// TIA Portal V17 export
// export: Created 2025-03-10T13:11:55.1694581Z, ExportSetting WithDefaults, DisplayName Totally Integrated Automation Portal, DisplayVersion V17 Update 8, DisplayName TIA Portal Openness, DisplayVersion V17 Update 8, DisplayName TIA Portal Version Control Interface, DisplayVersion V17, DisplayName SINAMICS Startdrive Advanced, DisplayVersion V17 SP2, DisplayName SINAMICS Startdrive G110M, G120, G120C, G120D, G120P, G115D, DisplayVersion V17 SP2, DisplayName SINAMICS Startdrive G130, G150, S120, S150, SINAMICS MV, S210, DisplayVersion V17 SP2, DisplayName STEP 7 Professional, DisplayVersion V17 Update 8, DisplayName SINUMERIK ONE STEP 7 Toolbox, DisplayVersion V17 Update 12, DisplayName SINUMERIK 840D sl STEP 7 Toolbox, DisplayVersion V17 Update 12, DisplayName STEP 7 Safety, DisplayVersion V17 Update 6, DisplayName WinCC Advanced, DisplayVersion V17 Update 8
TYPE "LBP_typeTMLoadMT"
TITLE = Tool management / Gestión de herramientas / Werkzeugverwaltung
// User data type for block LBP_TMLoadMT [DB1071] / Tipo de dato de usuario para bloque LBP_TMLoadMT [DB1071] / Anwender-Datentyp für Baustein LBP_TMLoadMT [DB1071]
// stored: IsFailsafeCompliant false
   STRUCT
      MTIF : Array[1..16] of Struct
         DistanceCoding : Int;   // Art der Entfernungscodierung ($TC_MTP_KD) / Type of distance coding ($TC_MTP_KD) / Tipo de codificación de distancia ($TC_MTP_KD)
         Places : Int;   // Anzahl der Plätze des Multitools / Number of locations of the multitool / Número de puestos de Multitool
         Distance : Real;   // Entfernung des Multitool-Platzes / Multitool location distance / Distancia a puesto Multitool
         MTNo : Int;   // Interne WZ-Nummer des Multitools / Internal T number of the multitool / Número de herramienta interno de Multitool
         PlaceNo : Int;   // Platznummer im Multitool, auf die das System positioniert / Location number within the multitool to which the system positions / Número de puesto de Multitool en el que posiciona el sistema
         Toolholder : Int;   // Spindel- oder Werkzeughalter-Nummer / Spindle or toolholder number / Número de cabezal o de portaherramientas
         reserved : Array[1..3] of Int;   // Reserviert / Reserved / Reservado
      END_STRUCT;
   END_STRUCT;
   // // MTIF[2].DistanceCoding : Art der Entfernungscodierung ($TC_MTP_KD) / Type of distance coding ($TC_MTP_KD) / Tipo de codificación de distancia ($TC_MTP_KD)
   // // MTIF[3].DistanceCoding : Art der Entfernungscodierung ($TC_MTP_KD) / Type of distance coding ($TC_MTP_KD) / Tipo de codificación de distancia ($TC_MTP_KD)
   // // MTIF[4].DistanceCoding : Art der Entfernungscodierung ($TC_MTP_KD) / Type of distance coding ($TC_MTP_KD) / Tipo de codificación de distancia ($TC_MTP_KD)
   // // MTIF[5].DistanceCoding : Art der Entfernungscodierung ($TC_MTP_KD) / Type of distance coding ($TC_MTP_KD) / Tipo de codificación de distancia ($TC_MTP_KD)
   // // MTIF[6].DistanceCoding : Art der Entfernungscodierung ($TC_MTP_KD) / Type of distance coding ($TC_MTP_KD) / Tipo de codificación de distancia ($TC_MTP_KD)
   // // MTIF[7].DistanceCoding : Art der Entfernungscodierung ($TC_MTP_KD) / Type of distance coding ($TC_MTP_KD) / Tipo de codificación de distancia ($TC_MTP_KD)
   // // MTIF[8].DistanceCoding : Art der Entfernungscodierung ($TC_MTP_KD) / Type of distance coding ($TC_MTP_KD) / Tipo de codificación de distancia ($TC_MTP_KD)
   // // MTIF[9].DistanceCoding : Art der Entfernungscodierung ($TC_MTP_KD) / Type of distance coding ($TC_MTP_KD) / Tipo de codificación de distancia ($TC_MTP_KD)
   // // MTIF[10].DistanceCoding : Art der Entfernungscodierung ($TC_MTP_KD) / Type of distance coding ($TC_MTP_KD) / Tipo de codificación de distancia ($TC_MTP_KD)
   // // MTIF[11].DistanceCoding : Art der Entfernungscodierung ($TC_MTP_KD) / Type of distance coding ($TC_MTP_KD) / Tipo de codificación de distancia ($TC_MTP_KD)
   // // MTIF[12].DistanceCoding : Art der Entfernungscodierung ($TC_MTP_KD) / Type of distance coding ($TC_MTP_KD) / Tipo de codificación de distancia ($TC_MTP_KD)
   // // MTIF[13].DistanceCoding : Art der Entfernungscodierung ($TC_MTP_KD) / Type of distance coding ($TC_MTP_KD) / Tipo de codificación de distancia ($TC_MTP_KD)
   // // MTIF[14].DistanceCoding : Art der Entfernungscodierung ($TC_MTP_KD) / Type of distance coding ($TC_MTP_KD) / Tipo de codificación de distancia ($TC_MTP_KD)
   // // MTIF[15].DistanceCoding : Art der Entfernungscodierung ($TC_MTP_KD) / Type of distance coding ($TC_MTP_KD) / Tipo de codificación de distancia ($TC_MTP_KD)
   // // MTIF[16].DistanceCoding : Art der Entfernungscodierung ($TC_MTP_KD) / Type of distance coding ($TC_MTP_KD) / Tipo de codificación de distancia ($TC_MTP_KD)
   // // MTIF[2].Places : Anzahl der Plätze des Multitools / Number of locations of the multitool / Número de puestos de Multitool
   // // MTIF[3].Places : Anzahl der Plätze des Multitools / Number of locations of the multitool / Número de puestos de Multitool
   // // MTIF[4].Places : Anzahl der Plätze des Multitools / Number of locations of the multitool / Número de puestos de Multitool
   // // MTIF[5].Places : Anzahl der Plätze des Multitools / Number of locations of the multitool / Número de puestos de Multitool
   // // MTIF[6].Places : Anzahl der Plätze des Multitools / Number of locations of the multitool / Número de puestos de Multitool
   // // MTIF[7].Places : Anzahl der Plätze des Multitools / Number of locations of the multitool / Número de puestos de Multitool
   // // MTIF[8].Places : Anzahl der Plätze des Multitools / Number of locations of the multitool / Número de puestos de Multitool
   // // MTIF[9].Places : Anzahl der Plätze des Multitools / Number of locations of the multitool / Número de puestos de Multitool
   // // MTIF[10].Places : Anzahl der Plätze des Multitools / Number of locations of the multitool / Número de puestos de Multitool
   // // MTIF[11].Places : Anzahl der Plätze des Multitools / Number of locations of the multitool / Número de puestos de Multitool
   // // MTIF[12].Places : Anzahl der Plätze des Multitools / Number of locations of the multitool / Número de puestos de Multitool
   // // MTIF[13].Places : Anzahl der Plätze des Multitools / Number of locations of the multitool / Número de puestos de Multitool
   // // MTIF[14].Places : Anzahl der Plätze des Multitools / Number of locations of the multitool / Número de puestos de Multitool
   // // MTIF[15].Places : Anzahl der Plätze des Multitools / Number of locations of the multitool / Número de puestos de Multitool
   // // MTIF[16].Places : Anzahl der Plätze des Multitools / Number of locations of the multitool / Número de puestos de Multitool
   // // MTIF[2].Distance : Entfernung des Multitool-Platzes / Multitool location distance / Distancia a puesto Multitool
   // // MTIF[3].Distance : Entfernung des Multitool-Platzes / Multitool location distance / Distancia a puesto Multitool
   // // MTIF[4].Distance : Entfernung des Multitool-Platzes / Multitool location distance / Distancia a puesto Multitool
   // // MTIF[5].Distance : Entfernung des Multitool-Platzes / Multitool location distance / Distancia a puesto Multitool
   // // MTIF[6].Distance : Entfernung des Multitool-Platzes / Multitool location distance / Distancia a puesto Multitool
   // // MTIF[7].Distance : Entfernung des Multitool-Platzes / Multitool location distance / Distancia a puesto Multitool
   // // MTIF[8].Distance : Entfernung des Multitool-Platzes / Multitool location distance / Distancia a puesto Multitool
   // // MTIF[9].Distance : Entfernung des Multitool-Platzes / Multitool location distance / Distancia a puesto Multitool
   // // MTIF[10].Distance : Entfernung des Multitool-Platzes / Multitool location distance / Distancia a puesto Multitool
   // // MTIF[11].Distance : Entfernung des Multitool-Platzes / Multitool location distance / Distancia a puesto Multitool
   // // MTIF[12].Distance : Entfernung des Multitool-Platzes / Multitool location distance / Distancia a puesto Multitool
   // // MTIF[13].Distance : Entfernung des Multitool-Platzes / Multitool location distance / Distancia a puesto Multitool
   // // MTIF[14].Distance : Entfernung des Multitool-Platzes / Multitool location distance / Distancia a puesto Multitool
   // // MTIF[15].Distance : Entfernung des Multitool-Platzes / Multitool location distance / Distancia a puesto Multitool
   // // MTIF[16].Distance : Entfernung des Multitool-Platzes / Multitool location distance / Distancia a puesto Multitool
   // // MTIF[2].MTNo : Interne WZ-Nummer des Multitools / Internal T number of the multitool / Número de herramienta interno de Multitool
   // // MTIF[3].MTNo : Interne WZ-Nummer des Multitools / Internal T number of the multitool / Número de herramienta interno de Multitool
   // // MTIF[4].MTNo : Interne WZ-Nummer des Multitools / Internal T number of the multitool / Número de herramienta interno de Multitool
   // // MTIF[5].MTNo : Interne WZ-Nummer des Multitools / Internal T number of the multitool / Número de herramienta interno de Multitool
   // // MTIF[6].MTNo : Interne WZ-Nummer des Multitools / Internal T number of the multitool / Número de herramienta interno de Multitool
   // // MTIF[7].MTNo : Interne WZ-Nummer des Multitools / Internal T number of the multitool / Número de herramienta interno de Multitool
   // // MTIF[8].MTNo : Interne WZ-Nummer des Multitools / Internal T number of the multitool / Número de herramienta interno de Multitool
   // // MTIF[9].MTNo : Interne WZ-Nummer des Multitools / Internal T number of the multitool / Número de herramienta interno de Multitool
   // // MTIF[10].MTNo : Interne WZ-Nummer des Multitools / Internal T number of the multitool / Número de herramienta interno de Multitool
   // // MTIF[11].MTNo : Interne WZ-Nummer des Multitools / Internal T number of the multitool / Número de herramienta interno de Multitool
   // // MTIF[12].MTNo : Interne WZ-Nummer des Multitools / Internal T number of the multitool / Número de herramienta interno de Multitool
   // // MTIF[13].MTNo : Interne WZ-Nummer des Multitools / Internal T number of the multitool / Número de herramienta interno de Multitool
   // // MTIF[14].MTNo : Interne WZ-Nummer des Multitools / Internal T number of the multitool / Número de herramienta interno de Multitool
   // // MTIF[15].MTNo : Interne WZ-Nummer des Multitools / Internal T number of the multitool / Número de herramienta interno de Multitool
   // // MTIF[16].MTNo : Interne WZ-Nummer des Multitools / Internal T number of the multitool / Número de herramienta interno de Multitool
   // // MTIF[2].PlaceNo : Platznummer im Multitool, auf die das System positioniert / Location number within the multitool to which the system positions / Número de puesto de Multitool en el que posiciona el sistema
   // // MTIF[3].PlaceNo : Platznummer im Multitool, auf die das System positioniert / Location number within the multitool to which the system positions / Número de puesto de Multitool en el que posiciona el sistema
   // // MTIF[4].PlaceNo : Platznummer im Multitool, auf die das System positioniert / Location number within the multitool to which the system positions / Número de puesto de Multitool en el que posiciona el sistema
   // // MTIF[5].PlaceNo : Platznummer im Multitool, auf die das System positioniert / Location number within the multitool to which the system positions / Número de puesto de Multitool en el que posiciona el sistema
   // // MTIF[6].PlaceNo : Platznummer im Multitool, auf die das System positioniert / Location number within the multitool to which the system positions / Número de puesto de Multitool en el que posiciona el sistema
   // // MTIF[7].PlaceNo : Platznummer im Multitool, auf die das System positioniert / Location number within the multitool to which the system positions / Número de puesto de Multitool en el que posiciona el sistema
   // // MTIF[8].PlaceNo : Platznummer im Multitool, auf die das System positioniert / Location number within the multitool to which the system positions / Número de puesto de Multitool en el que posiciona el sistema
   // // MTIF[9].PlaceNo : Platznummer im Multitool, auf die das System positioniert / Location number within the multitool to which the system positions / Número de puesto de Multitool en el que posiciona el sistema
   // // MTIF[10].PlaceNo : Platznummer im Multitool, auf die das System positioniert / Location number within the multitool to which the system positions / Número de puesto de Multitool en el que posiciona el sistema
   // // MTIF[11].PlaceNo : Platznummer im Multitool, auf die das System positioniert / Location number within the multitool to which the system positions / Número de puesto de Multitool en el que posiciona el sistema
   // // MTIF[12].PlaceNo : Platznummer im Multitool, auf die das System positioniert / Location number within the multitool to which the system positions / Número de puesto de Multitool en el que posiciona el sistema
   // // MTIF[13].PlaceNo : Platznummer im Multitool, auf die das System positioniert / Location number within the multitool to which the system positions / Número de puesto de Multitool en el que posiciona el sistema
   // // MTIF[14].PlaceNo : Platznummer im Multitool, auf die das System positioniert / Location number within the multitool to which the system positions / Número de puesto de Multitool en el que posiciona el sistema
   // // MTIF[15].PlaceNo : Platznummer im Multitool, auf die das System positioniert / Location number within the multitool to which the system positions / Número de puesto de Multitool en el que posiciona el sistema
   // // MTIF[16].PlaceNo : Platznummer im Multitool, auf die das System positioniert / Location number within the multitool to which the system positions / Número de puesto de Multitool en el que posiciona el sistema
   // // MTIF[2].Toolholder : Spindel- oder Werkzeughalter-Nummer / Spindle or toolholder number / Número de cabezal o de portaherramientas
   // // MTIF[3].Toolholder : Spindel- oder Werkzeughalter-Nummer / Spindle or toolholder number / Número de cabezal o de portaherramientas
   // // MTIF[4].Toolholder : Spindel- oder Werkzeughalter-Nummer / Spindle or toolholder number / Número de cabezal o de portaherramientas
   // // MTIF[5].Toolholder : Spindel- oder Werkzeughalter-Nummer / Spindle or toolholder number / Número de cabezal o de portaherramientas
   // // MTIF[6].Toolholder : Spindel- oder Werkzeughalter-Nummer / Spindle or toolholder number / Número de cabezal o de portaherramientas
   // // MTIF[7].Toolholder : Spindel- oder Werkzeughalter-Nummer / Spindle or toolholder number / Número de cabezal o de portaherramientas
   // // MTIF[8].Toolholder : Spindel- oder Werkzeughalter-Nummer / Spindle or toolholder number / Número de cabezal o de portaherramientas
   // // MTIF[9].Toolholder : Spindel- oder Werkzeughalter-Nummer / Spindle or toolholder number / Número de cabezal o de portaherramientas
   // // MTIF[10].Toolholder : Spindel- oder Werkzeughalter-Nummer / Spindle or toolholder number / Número de cabezal o de portaherramientas
   // // MTIF[11].Toolholder : Spindel- oder Werkzeughalter-Nummer / Spindle or toolholder number / Número de cabezal o de portaherramientas
   // // MTIF[12].Toolholder : Spindel- oder Werkzeughalter-Nummer / Spindle or toolholder number / Número de cabezal o de portaherramientas
   // // MTIF[13].Toolholder : Spindel- oder Werkzeughalter-Nummer / Spindle or toolholder number / Número de cabezal o de portaherramientas
   // // MTIF[14].Toolholder : Spindel- oder Werkzeughalter-Nummer / Spindle or toolholder number / Número de cabezal o de portaherramientas
   // // MTIF[15].Toolholder : Spindel- oder Werkzeughalter-Nummer / Spindle or toolholder number / Número de cabezal o de portaherramientas
   // // MTIF[16].Toolholder : Spindel- oder Werkzeughalter-Nummer / Spindle or toolholder number / Número de cabezal o de portaherramientas
   // // MTIF[2].reserved : Reserviert / Reserved / Reservado
   // // MTIF[3].reserved : Reserviert / Reserved / Reservado
   // // MTIF[4].reserved : Reserviert / Reserved / Reservado
   // // MTIF[5].reserved : Reserviert / Reserved / Reservado
   // // MTIF[6].reserved : Reserviert / Reserved / Reservado
   // // MTIF[7].reserved : Reserviert / Reserved / Reservado
   // // MTIF[8].reserved : Reserviert / Reserved / Reservado
   // // MTIF[9].reserved : Reserviert / Reserved / Reservado
   // // MTIF[10].reserved : Reserviert / Reserved / Reservado
   // // MTIF[11].reserved : Reserviert / Reserved / Reservado
   // // MTIF[12].reserved : Reserviert / Reserved / Reservado
   // // MTIF[13].reserved : Reserviert / Reserved / Reservado
   // // MTIF[14].reserved : Reserviert / Reserved / Reservado
   // // MTIF[15].reserved : Reserviert / Reserved / Reservado
   // // MTIF[16].reserved : Reserviert / Reserved / Reservado
END_TYPE
